# EPICS autosave request: dxpApp/Db/dxpHighLevel_settings.req
$(P)$(R)DetectionThreshold
$(P)$(R)MinPulsePairSeparation
$(P)$(R)DetectionFilter
$(P)$(R)ScaleFactor
$(P)$(R)DetectorPolarity
$(P)$(R)DecayTime
$(P)$(R)PresetMode
$(P)$(R)PresetEvents
$(P)$(R)PresetTriggers
